Yaskawa INFORM job: READTWS_B.JBI

/JOB
//NAME READTWS_B
///FOLDERNAME MASTER
//POS
///NPOS 0,0,0,0,0,0
//INST
///DATE 2021/10/29 11:49
///ATTR SC,RO
NOP
'*****************************
'READ THE RIGHT TWO DIGITS OF
'TWS AND SET IN B020.
'*****************************
DOUT OT#(18) OFF
DOUT OT#(19) OFF
DOUT OT#(20) OFF
DOUT OT#(17) ON
TIMER T=0.20
DIN B020 IGH#(5)
TIMER T=0.10
DOUT OT#(17) OFF
DOUT OT#(18) ON
TIMER T=0.20
DIN B021 IGH#(5)
TIMER T=0.10
DOUT OT#(18) OFF
MUL B021 10
ADD B020 B021
END
